// TIA Portal V17 export
// export: Created 2025-03-05T08:02:40.2635698Z, ExportSetting WithDefaults, DisplayName Totally Integrated Automation Portal, DisplayVersion V17 Update 8, DisplayName TIA Portal Openness, DisplayVersion V17 Update 8, DisplayName TIA Portal Version Control Interface, DisplayVersion V17, DisplayName SINAMICS Startdrive Advanced, DisplayVersion V17 SP2, DisplayName SINAMICS Startdrive G110M, G120, G120C, G120D, G120P, G115D, DisplayVersion V17 SP2, DisplayName SINAMICS Startdrive G130, G150, S120, S150, SINAMICS MV, S210, DisplayVersion V17 SP2, DisplayName STEP 7 Professional, DisplayVersion V17 Update 8, DisplayName SINUMERIK ONE STEP 7 Toolbox, DisplayVersion V17 Update 12, DisplayName SINUMERIK 840D sl STEP 7 Toolbox, DisplayVersion V17 Update 12, DisplayName STEP 7 Safety, DisplayVersion V17 Update 6, DisplayName WinCC Advanced, DisplayVersion V17 Update 8
FUNCTION "FC428_OPERATOR_HELP" : Void   // FC428, LAD
{ S7_Optimized_Access := 'FALSE' }
AUTHOR : ETXETAR
VERSION : 1.0
// stored: AutoNumber false, IsIECCheckEnabled false, SetENOAutomatically false, UDAEnableTagReadback false
   VAR_TEMP
      Byte_Number : Int;
      Help_Number : Int;
      Part_Type : Int;
   END_VAR
BEGIN

NETWORK
TITLE = OPERATOR HELP
      LAR1  P#0.0;
      L     0;
      T     #Help_Number;
      L     1000;
M001: T     #Byte_Number;
      OPN   "DB428_OPERATOR_HELP";
      L     #Help_Number;
      L     1;
      +I;
      T     #Help_Number;
      A     DBX [AR1, P#0.1];
      JC    M002;
      +AR1  P#0.1;
      L     #Byte_Number;
      LOOP  M001;
M002: L     #Help_Number;
      T     "DB2000_WINCC_HMI_FUNCTION".HELP_PROMPT;



REGION Network 2: OPERATOR HELP RESET
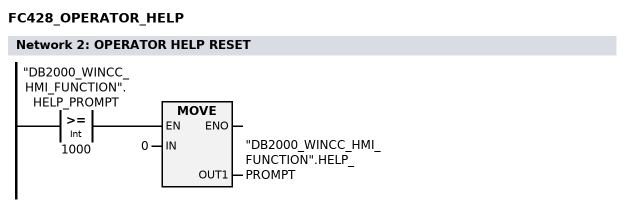
   RUNG wire#powerrail
      { S7_Templates := "SrcType := Int" } GE_Contact(in1 := "DB2000_WINCC_HMI_FUNCTION".HELP_PROMPT, in2 := 1000)
      Move(in := 0, out1 => "DB2000_WINCC_HMI_FUNCTION".HELP_PROMPT)
   END_RUNG
   // the same network as SCL:
   IF "DB2000_WINCC_HMI_FUNCTION".HELP_PROMPT >= 1000 THEN
       "DB2000_WINCC_HMI_FUNCTION".HELP_PROMPT := 0;
   END_IF;
END_REGION
END_FUNCTION
